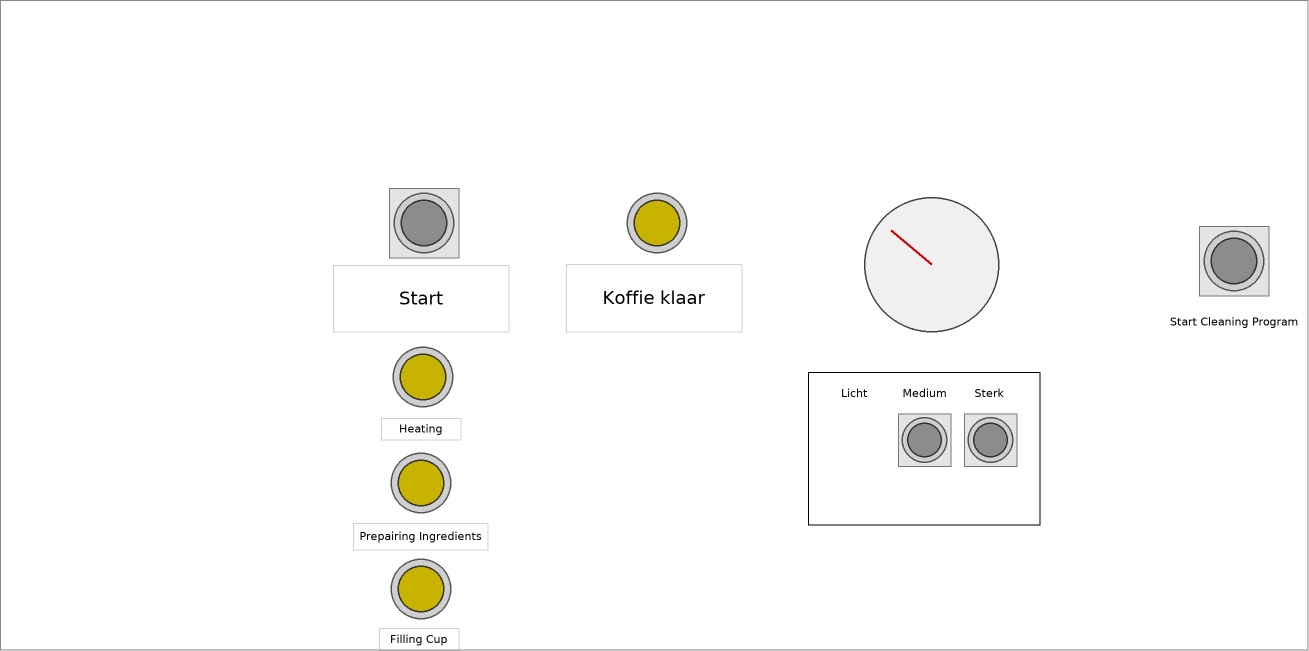
VISUALIZATION Visualization  // 1309x651
    Lamp1 (388,342 70x70), variable: Heating.Heating, style: Lamp-Lamp1-Yellow
    Lamp1 (386,448 70x70), variable: Prepare_Ingredients.Prepairing, style: Lamp-Lamp1-Yellow
    PushSwitchLed (389,188 70x70), variable: GVL.Start, behaviour: TOGGLE, style: Switch-PushSwitchLed-Gray
    Textfield (333,265 176x67), "Start"
    Textfield (381,418 80x22), "Heating"
    Textfield (353,523 135x27), "Prepairing Ingredients"
    Lamp1 (622,188 70x70), variable: Fill_Cup.Ready, style: Lamp-Lamp1-Yellow
    Textfield (566,264 176x68), "Koffie klaar"
    Meter180 (788,197 287x135), value: Heating.WaterTemp, style: Meter-Meter180-Yellow, scale format: %.1f, scale 0..100
        p518627256: Watertemperatuur
    Lamp1 (386,554 70x70), variable: Fill_Cup.Filling, style: Lamp-Lamp1-Yellow
    Textfield (379,628 80x23), "Filling Cup"
    Lamp1 (840,473 41x38), variable: Lamp_Loop.Lamp1, style: Lamp-Lamp1-Yellow
    Lamp1 (907,473 41x38), variable: Lamp_Loop.Lamp2, style: Lamp-Lamp1-Yellow
    Lamp1 (972,473 41x38), variable: Lamp_Loop.Lamp3, style: Lamp-Lamp1-Yellow
    Frame (979,444 1x0)
    PushSwitch (832,410 53x60), variable: Fill_Cup.Licht, behaviour: TOGGLE, style: Switch-PushSwitch-Gray
    Rectangle (808,372 232x153)
    Textfield (813,378 219x31), "Licht Medium Sterk"
    PushSwitch (898,410 53x60), variable: Fill_Cup.Medium, behaviour: TOGGLE, style: Switch-PushSwitch-Gray
    PushSwitch (964,410 53x60), variable: Fill_Cup.Sterk, behaviour: TOGGLE, style: Switch-PushSwitch-Gray
    PushSwitch (1199,226 70x70), variable: GVL.CleanMachine, behaviour: TOGGLE, style: Switch-PushSwitch-Gray
    Label (1159,307 150x30), "Start Cleaning Program"
END_VISUALIZATION

(* stored: Version 1.1.0.1, ProductVersion 3.1.4024.12
   Visu Visualization: Id {f5b13e13-4582-4db1-911a-c2d252b43be6} *)
